// Mitsubishi GX Works2 project: Test   PLC: FX1N/FX1NC

TYPE Axis : STRUCT
  CurFS : DINT;  (* int Current feed speed *)
  Dir : BOOL;  (* bool Direction *)
  DirInt : DINT;  (* int Direction *)
  Limited : BOOL;  (* bool Limit reached *)
  CurPos : DINT;  (* int Current position (mm) *)
  CurPosP : DINT;  (* int Current position (pulse) *)
  TarFS : DINT;  (* int Target feed speed *)
  TarPos : DINT;  (* int Target position (mm) *)
  TarPosP : DINT;  (* int Target position (pulse) *)
  ManualN : BOOL;  (* bool Manual run: Negative direction *)
  ManualP : BOOL;  (* bool Manual run: Possitive direction *)
  ILimitN : BOOL;
  ILimitP : BOOL;
  OOnOff : BOOL;
  OReset : BOOL;
  OPulse : BOOL;
  ODirection : BOOL;
  TarR : BOOL;  (* bool Target reached *)
END_STRUCT END_TYPE

// global labels: Global1
VAR_GLOBAL
  OriginSetMove : OriginSetMove;
  IsOn AT M0 : BOOL;
  ResetButton AT M2 : BOOL;
  StopButton AT M9 : BOOL;
  SetButton AT M5 : BOOL;
  OriginButton AT M7 : BOOL;
  OnOffResetStop : OnOffResetStop;
  TargetReached : BOOL;
  CommandLt : INT;
  CommandNb : INT;
  OLazer AT Y004 : BOOL;
  ArrayEnded AT M11 : BOOL;
  AutoNextLine AT M10 : BOOL;
  ArrayIndex AT D10 : INT;
  ArrayIndexMax AT D11 : INT;
  XX : Axis;
  ManualHandler : ManualHandler;
  YY : Axis;
  RunStart : BOOL;
  RunNext : BOOL;
  RunButton AT M8 : BOOL;
  FeedSpeed AT D0 : DINT;
END_VAR

// task Task_01 (event TRUE, interval 0, priority 31): POU_01

PROGRAM POU_01
VAR
  fRunLatchY : BOOL;
END_VAR
OnOffResetStop();

IF IsOn THEN
	ManualHandler();
	
	SET(RunButton OR RunNext, RunStart);
	IF RunStart THEN
		XX.TarPosP := XX.TarPos;
		XX.TarR := XX.CurPosP >= XX.TarPosP;
		DMOV(NOT XX.TarR, FeedSpeed, XX.CurFS);
		YY.TarPosP := YY.TarPos;
		YY.TarR := YY.CurPosP >= YY.TarPosP;
		DMOV(NOT YY.TarR, FeedSpeed, YY.CurFS);
		
		TargetReached := XX.TarR AND YY.TarR;
		RunNext := FALSE;
	END_IF;
	
	DPLSV(TRUE, XX.CurFS, XX.OPulse, XX.Dir);
	OUT(NOT XX.Dir, XX.ODirection);
	DPLSV(TRUE, YY.CurFS, YY.OPulse, YY.Dir);
	OUT(NOT YY.Dir, YY.ODirection);

	SET(XX.CurPosP >= YY.TarPosP, XX.TarR);
	RST(XX.TarR, XX.CurFS);
	SET(YY.CurPosP >= YY.TarPosP, YY.TarR);
	RST(YY.TarR, YY.CurFS);
	SET(XX.TarR AND YY.TarR, TargetReached);

	IF TargetReached AND AutoNextLine THEN
		YY.TarPos := YY.TarPos + INT_TO_DINT(ArrayIndex);
		SET(YY.TarPos <= 20000, RunNext);
		RST(NOT RunNext, YY.CurFS);
		RST(NOT RunNext, AutoNextLine);
	END_IF;
	TargetReached := FALSE;
	
	RunStart := FALSE;
	RunButton := FALSE;
	XX.CurPos := XX.CurPosP;
	YY.CurPos := YY.CurPosP;
			
	OriginSetMove();
END_IF;
END_PROGRAM

FUNCTION_BLOCK OnOffResetStop
OUT(IsOn, XX.OOnOff);
OUT(IsOn, YY.OOnOff);

SET(ResetButton, XX.OReset);
SET(ResetButton, YY.OReset);
OUT_T(ResetButton, TC200, 8);
RST(TC200, ResetButton);
RST(TC200, XX.OReset);
RST(TC200, YY.OReset);

RST(StopButton, RunButton);
RST(StopButton, ArrayEnded);
RST(StopButton, AutoNextLine);
RST(StopButton, TargetReached);
RST(StopButton, StopButton);
END_FUNCTION_BLOCK

FUNCTION_BLOCK OriginSetMove
VAR
  SetOrigin : BOOL;
  MoveToOrigin : BOOL;
END_VAR
OUT(OriginButton AND SetButton, SetOrigin);
OUT(OriginButton AND NOT SetButton, MoveToOrigin);

RST(SetOrigin, XX.CurPos);
RST(SetOrigin, XX.CurPosP);
RST(SetOrigin, YY.CurPos);
RST(SetOrigin, YY.CurPosP);
RST(SetOrigin, SetButton);

RST(MoveToOrigin, XX.TarPos);
RST(MoveToOrigin, XX.TarPosP);
RST(MoveToOrigin, YY.TarPos);
RST(MoveToOrigin, YY.TarPosP);
SET(MoveToOrigin, RunButton);

RST(SetOrigin OR MoveToOrigin, OriginButton);
END_FUNCTION_BLOCK

FUNCTION_BLOCK ManualHandler
IF NOT (RunButton OR AutoNextLine) THEN
	OUT((NOT XX.ILimitN AND XX.ManualN) OR (NOT XX.ILimitP AND XX.ManualP), XX.Limited);
	DMOV(NOT XX.Limited AND XX.ManualN, -FeedSpeed, XX.CurFS);
	DMOV(NOT XX.Limited AND XX.ManualP, FeedSpeed, XX.CurFS);
	RST(XX.Limited, XX.CurFS);
	
	OUT((NOT YY.ILimitN AND YY.ManualN) OR (NOT YY.ILimitP AND YY.ManualP), YY.Limited);
	DMOV(NOT YY.Limited AND YY.ManualN, -FeedSpeed, YY.CurFS);
	DMOV(NOT YY.Limited AND YY.ManualP, FeedSpeed, YY.CurFS);
	RST(YY.Limited, YY.CurFS);
END_IF;
END_FUNCTION_BLOCK
